TYPE AppConfig :
STRUCT
	NetIdManagement : NetIdManagement;
	CanOverEthercatConfig : CanOverEthercatConfig;
	LogConfig : LogConfig;
	CalibrateConfig : CalibrateConfig;
END_STRUCT
END_TYPE

(* stored: Version 1.1.0.1, ProductVersion 3.1.4024.12
   DUT AppConfig: Id {b9ac9a44-b964-4d40-9fe2-0ca20efb7a6c} *)
